Fanuc KAREL source: ko00083.KL

-- PROVISIONAL review KL for V1013-1; original PC SHA256 b537e58a6fdd6b640b3eb6447485922e517fdf2e737fc882aca2869516df5b48
-- Incomplete behavior may be omitted. Consult companion uncertainty JSON. Do not deploy.
PROGRAM KO00083
%NOLOCKGROUP
BEGIN
  -- UNRESOLVED_PC offsets 5-12; opcodes 9D,23
  -- UNRESOLVED_PC offsets 17-66; opcodes 27,27,49,7E,AD,22,1C,22,31,7E,4A
  -- UNRESOLVED_PC offsets 71-75; opcodes 7F
END KO00083
